{attribute 'GeneratedUsingTerminal: EL3446-0000-0016'}
{attribute addProperty BoxType "EL3446-0000-0016"}
{attribute addProperty Id "I1_CurrentAT %I*I1_Current_AFE1DFA29I2_CurrentAT %I*I2_Current_AFE1DFA29I3_CurrentAT %I*I3_Current_AFE1DFA29I4_CurrentAT %I*I4_Current_AFE1DFA29I5_CurrentAT %I*I5_Current_AFE1DFA29I6_CurrentAT %I*I6_Current_AFE1DFA29WcStateAT %I*WcState_9091E0EB2InfoDataAT %I*InfoData_1088C70510"}
{attribute addProperty CRC "1343575244"}
{attribute addProperty Size "66"}
TYPE EL3446_501554CC EXTENDS EtcSlaveTerminalBase_947E5A46 :
STRUCT
	{attribute addProperty Name "I1_Current"}
	I1_Current : I1_Current_AFE1DFA2;
	{attribute addProperty Name "I2_Current"}
	I2_Current : I2_Current_AFE1DFA2;
	{attribute addProperty Name "I3_Current"}
	I3_Current : I3_Current_AFE1DFA2;
	{attribute addProperty Name "I4_Current"}
	I4_Current : I4_Current_AFE1DFA2;
	{attribute addProperty Name "I5_Current"}
	I5_Current : I5_Current_AFE1DFA2;
	{attribute addProperty Name "I6_Current"}
	I6_Current : I6_Current_AFE1DFA2;
	{attribute addProperty Name "WcState"}
	WcState : WcState_9091E0EB;
	{attribute addProperty Name "InfoData"}
	InfoData : InfoData_1088C705;
END_STRUCT
END_TYPE

(* stored: Version 1.2.0.0, ProductVersion 3.1.4024.9
   DUT EL3446_501554CC: Id {74f0ade8-76b3-4ec3-82ee-ac1207ed554b} *)
